(* PLC project plc_copy, Dassault Systèmes ControlBuild 2024x Refresh1 *)
(* stored: creationDateTime 2024-04-15T11:44:30-01:00 *)

PROGRAM flask_motion_app.plc_copy

(* FBD diagram, written out as Structured Text *)
END_PROGRAM
